TYPE ST_AxisStopParameter :
STRUCT
	fDeceleration: LREAL;
	fJerk: LREAL;
	fGap: LREAL;
	stOptions: ST_MoveOptions;
END_STRUCT
END_TYPE

(* stored: Version 1.1.0.1, ProductVersion 3.1.4022.18
   DUT ST_AxisStopParameter: Id {4f232219-e572-487f-9b1e-03dfb79ded44} *)
